FUNCTION_BLOCK MyBlock
  (* Standard: 61499-2 *)
  (* Version 1.0, 2026-06-15, Dimitrios Kalligaridis *)
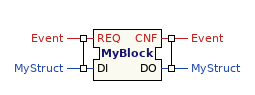
  EVENT_INPUT
    REQ WITH DI;
  END_EVENT
  EVENT_OUTPUT
    CNF WITH DO;
  END_EVENT
  VAR_INPUT
    DI : mypackage::MyStruct;
  END_VAR
  VAR_OUTPUT
    DO : mypackage::MyStruct;
  END_VAR
END_FUNCTION_BLOCK
